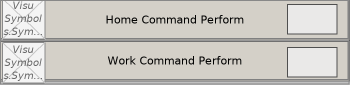
VISUALIZATION vActuatorFrame  // 350x85
VAR_INPUT
	iTextIndex1 : INT;
	iTextIndex2 : INT;
END_VAR
VAR_IN_OUT
	fbActuator:FB_ActuatorOOP_TC;
END_VAR
    Rectangle (0,0 350x81)
    Button (0,0 350x40), "Home Command Perform", pressed state: fbActuator.bHomeCmd, input disabled if: NOT fbActuator.bManualMode OR NOT fbActuator.prAllowHome, text list: 'tlActuatorNames', text index: iTextIndex1
        OnMouseClick: execute { fbActuator.mGoToHome(TRUE); }
    Button (0,41 350x40), "Work Command Perform", pressed state: fbActuator.bWorkCmd, input disabled if: NOT fbActuator.bManualMode OR NOT fbActuator.prAllowWork, text list: 'tlActuatorNames', text index: iTextIndex2
        OnMouseClick: execute { fbActuator.mGoToWork(TRUE); }
    Image (2,42 43x41), invisible if: fbActuator.prAllowWork, image: VisuSymbols.Symbols.Lock
    Image (2,-2 43x41), invisible if: fbActuator.prAllowHome, image: VisuSymbols.Symbols.Lock
    Rectangle (287,4 50x30), colour toggle: fbActuator.prInHomePosition
    Rectangle (287,47 50x30), colour toggle: fbActuator.prInWorkPosition
END_VISUALIZATION

(* stored: Version 1.1.0.1, ProductVersion 3.1.4024.15
   Visu vActuatorFrame: Id {a49e921c-8a0f-4cf3-8dff-74d4448b6a24} *)
